// TIA Portal V20 export
DATA_BLOCK "CallEquipment_DB"   // DB119
{ DB_Accessible_From_OPC_UA := 'FALSE' }
// stored: AssignedProDiagFB Unit1.Em11.ProDiag, DBAccessibleFromOPCUA false, DBAccessibleFromWebserver false, InstanceOfName Unit1.Em11.CallEquipment, InstanceOfType FB, Namespace Unit1.Em11
"Unit1.Em11.CallEquipment"
   // VAR_INPUT
   //    ZoneOperationEnable { ExternalWritable := 'False'} : "LWONIK_typeSafetyZoneManualOperation";
   // END_VAR
   // VAR_IN_OUT
   //    unitStatus : "LAF_typeUnitStatus";
   //    emFeedback : "LUC_typeEmFeedback";
   //    unitAlarmDB : "LAF_typeAlarms";
   // END_VAR
   // VAR
   //    InstWeightCheckSequence { ExternalWritable := 'False'} : "Unit1.Em11.Sequence_1_WeightCheck";
   //    instWeightCheckHomeJob1 { ExternalWritable := 'False'} : "LAF_SelectJob";
   //    instWeightCheckLoadJob2 { ExternalWritable := 'False'} : "LAF_SelectJob";
   //    instWeightCheckInspectionJob3 { ExternalWritable := 'False'} : "LAF_SelectJob";
   //    instWeightCheckUnloadJob4 { ExternalWritable := 'False'} : "LAF_SelectJob";
   //    instCmWeightCheckJRDetect { ExternalWritable := 'False'} : "LBC_DigitalSignalCn";
   //    instWeightCheckControl { ExternalWritable := 'False'} : "LER_WeightCheck";
   //    instWeightCheckHistory { ExternalWritable := 'False'} : "LER_weightCheckHistory";
   //    instManageAlarms { ExternalWritable := 'False'} : "LAF_ManageAlarms";
   //    instEventsPFE { ExternalWritable := 'False'} : "Unit1.Em11.EventsPFE";
   //    statUnitStatus { ExternalWritable := 'False'} : "LAF_typeUnitStatus";
   //    statPartData { ExternalWritable := 'False'} : "LER_typePartData";
   //    statDataDelete { ExternalWritable := 'False'} : "LER_typePartData";
   //    statHistoryDeleteData { ExternalWritable := 'False'} : "LER_typeWeightCheckHistory";
   //    statRoutingOk { ExternalWritable := 'False'} : Array[0..99] of Bool;
   //    statRoutingNok { ExternalWritable := 'False'} : Array[0..99] of Bool;
   //    statHomeCheck { ExternalWritable := 'False'} : Array[0..99] of Bool;
   //    statTonTime { ExternalWritable := 'False'} : Array[0..999] of TON_TIME;
   //    statTofTime { ExternalWritable := 'False'} : Array[0..9] of TOF_TIME;
   //    statPulse { ExternalWritable := 'False'} : Array[0..999] of Bool;
   //    statEnableManualCmds { ExternalWritable := 'False'} : Bool;
   //    statNomalMode { ExternalWritable := 'False'} : Bool;
   //    citi_Ptrig : Array[0..20] of Bool;
   //    citiTon : Array[0..20] of TON_TIME;
   //    citi : Time;
   //    citiTest : Array[0..20] of Bool;
   //    instPFERecipe { S7_SetPoint := 'True'} : "Unit1.Em11.EventsPFE_Recipe";
   // END_VAR
BEGIN
END_DATA_BLOCK
